Omron CX-Programmer project НовыйПроект (CX-Programmer 9.52)

# PLC НовыйПЛК1: CP1L-E EM

## Global symbols (name address type ; comment)
AbsoluteCounterPoisition D30 DINT  ; Абсолютное значение счетчика импульсов энкодера
AnalogSP D101 CHANNEL  ; Задание скорости с платы аналоговых выходов ПЛК
D1000 CHANNEL  ; выбор адреса ПЧ
D1002 CHANNEL  ; Выбор типа ПЧ - МХ2
T0000 BOOL  ; Бит запуска преобразования в аналоговую форму
AutomaticControl W0.09 BOOL  ; Автоматическое управление
CounterMinDistanceBetweenSaws D42 DINT  ; Минимальное расстояние между пилами в импульсах энкодера
DecButton W18.01 BOOL  ; Кнопка декремента на панели
EndOfCycleInAutomatic W0.13 BOOL  ; Конец цикла автоматического режима
ForwardCommand 100.02 BOOL  ; Команда Вперед на ПЧ
IncButton W18.00 BOOL  ; Кнопка инкремента на панели
InverterReady 0.06 BOOL  ; Частотный преобразователь готов (сигнал с ПЧ)
InverterRunning 0.07 BOOL  ; Частотный преобразователь запущен (сигнал с ПЧ)
LeftLimitSwitch 0.08 BOOL  ; Левый концевик
ManualControl W0.04 BOOL  ; Ручное управление
ManualLeft W0.07 BOOL  ; Влево в ручном режиме
ManualRight W0.08 BOOL  ; Вправо в ручном режиме
MinDistanceBetweenSaws D40 DINT  ; Уставка минимального расстояния между пилами (в крайнем положении)
MoveToPosition W0.03 BOOL  ; Переехать в заданное положение
PID_control1 CoordinateConverting
PV_HighspeedCounter D35 DINT  ; Текущее значение высокоскоростного счетчика
PreviousCounterPosition D32 DINT  ; Предыдущая позиция энкодера
PulseTravelDistance W13 UDINT  ; Число импульсов, необходимое для достижения положения
PulseVelocityInManual W10 UDINT  ; Скорость выдачи импульсов в ручном режиме
ResetPositioningInAutomatic W0.12 BOOL  ; Сброс функции позиционирования из автоматического режима
ResetPositioningInManual W0.11 BOOL  ; Сброс функции позиционирования из ручного режима
ReverseCommand 100.03 BOOL  ; Команда Назад на ПЧ
RightLimitSwitch 0.03 BOOL  ; Правый концевик
SawInLimitPosition W0.06 BOOL  ; Пила в конечном положении
SawSetPosition D11 INT  ; Заданное положение пилы (мм)
SawTravelDirection W0.10 BOOL  ; Направление движения пилы
StartLeftButton W0.00 BOOL  ; $?St$Bk?_#[3] / Кнопка "Пуск влево"$?St$Bk?_#[3]
StartRightButton W0.01 BOOL  ; $?St$Bk?_#[4] / Кнопка "Пуск вправо"$?St$Bk?_#[4]
StopButton W0.02 BOOL  ; $?St$Bk?_#[5] / Кнопка "Стоп"$?St$Bk?_#[5]
SystemReady W0.05 BOOL  ; Система в норме
ПЧ INV002_Refresh_X31_

## Program НоваяЗадача1 (cyclic task 0)
Local symbols
SawTravelDirection1 W0.15 BOOL
UPRmax D200 DINT  ; ограничение управления
Пуск 110.00 BOOL
Реверс 110.01 BOOL

### Section hmi

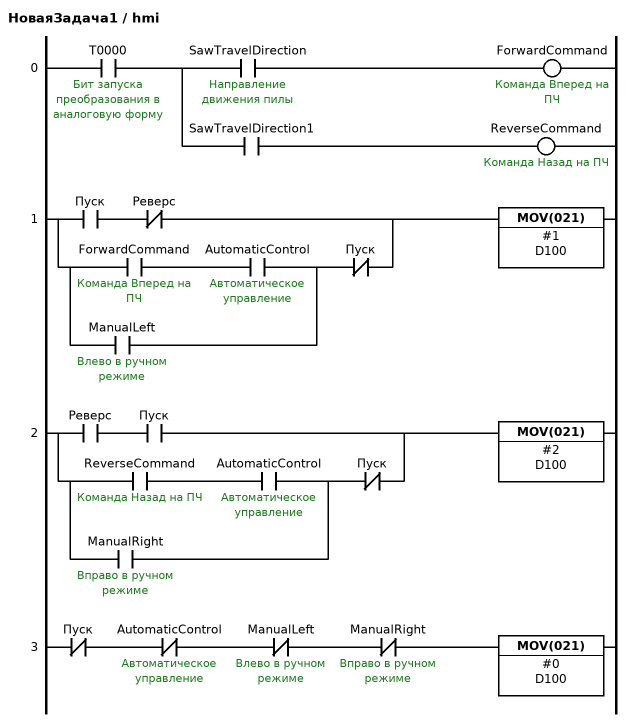
; rung 0
LD T0000  ; Бит запуска преобразования в аналоговую форму
OUT TR0
AND SawTravelDirection  ; Направление движения пилы
OUT ForwardCommand  ; Команда Вперед на ПЧ
LD TR0
AND SawTravelDirection1
OUT ReverseCommand  ; Команда Назад на ПЧ
; rung 1
LD Пуск
ANDNOT Реверс
LD ForwardCommand  ; Команда Вперед на ПЧ
AND AutomaticControl  ; Автоматическое управление
OR ManualLeft  ; Влево в ручном режиме
ANDNOT Пуск
ORLD
MOV(021) #1 D100
; rung 2
LD Реверс
AND Пуск
LD ReverseCommand  ; Команда Назад на ПЧ
AND AutomaticControl  ; Автоматическое управление
OR ManualRight  ; Вправо в ручном режиме
ANDNOT Пуск
ORLD
MOV(021) #2 D100
; rung 3
LDNOT Пуск
ANDNOT AutomaticControl  ; Автоматическое управление
ANDNOT ManualLeft  ; Влево в ручном режиме
ANDNOT ManualRight  ; Вправо в ручном режиме
MOV(021) #0 D100

### Section ModBus

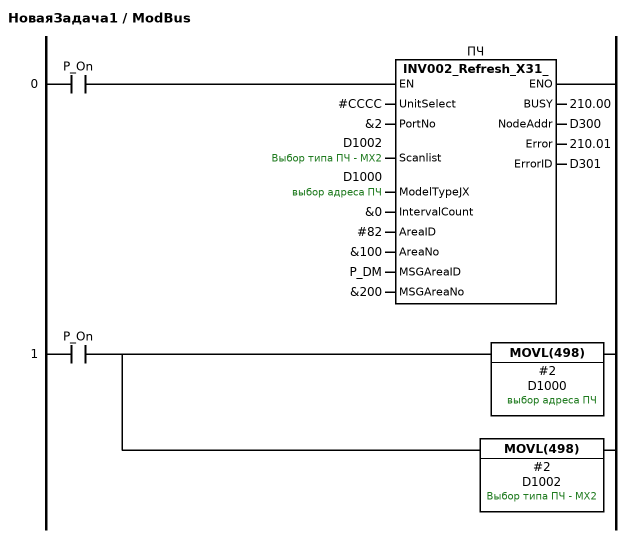
; rung 0
LD P_On
CALL ПЧ : INV002_Refresh_X31_ (UnitSelect := #CCCC, PortNo := &2, Scanlist := D1002, ModelTypeJX := D1000, IntervalCount := &0, AreaID := #82, AreaNo := &100, MSGAreaID := P_DM, MSGAreaNo := &200, BUSY => 210.00, NodeAddr => D300, Error => 210.01, ErrorID => D301)  ; Выбор типа ПЧ - МХ2, выбор адреса ПЧ
; rung 1
LD P_On
MOVL(498) #2 D1000  ; выбор адреса ПЧ
MOVL(498) #2 D1002  ; Выбор типа ПЧ - МХ2

### Section Initialization

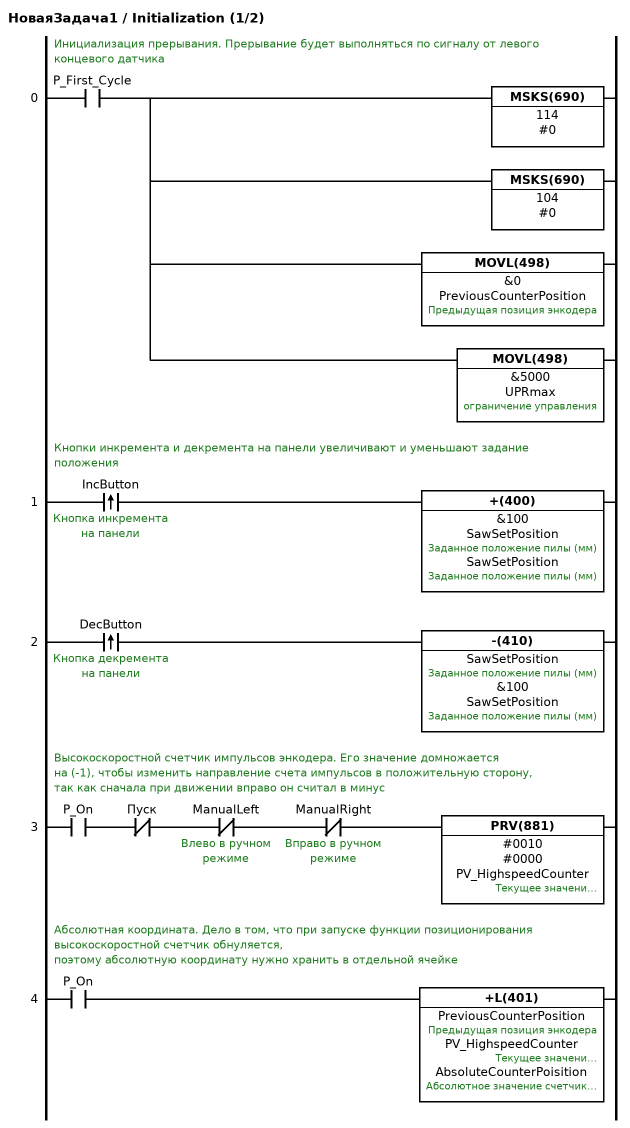
; rung 0: Инициализация прерывания. Прерывание будет выполняться по сигналу от левого концевого датчика
LD P_First_Cycle
MSKS(690) 114 #0
MSKS(690) 104 #0
MOVL(498) &0 PreviousCounterPosition  ; Предыдущая позиция энкодера
MOVL(498) &5000 UPRmax  ; ограничение управления
; rung 1: Кнопки инкремента и декремента на панели увеличивают и уменьшают задание положения
@LD IncButton  ; Кнопка инкремента на панели
+(400) &100 SawSetPosition SawSetPosition  ; Заданное положение пилы (мм)
; rung 2
@LD DecButton  ; Кнопка декремента на панели
-(410) SawSetPosition &100 SawSetPosition  ; Заданное положение пилы (мм)
; rung 3: Высокоскоростной счетчик импульсов энкодера. Его значение домножается / на (-1), чтобы изменить направление счета импульсов в положительную сторону, / так как сначала при движении вправо он считал в минус
LD P_On
ANDNOT Пуск
ANDNOT ManualLeft  ; Влево в ручном режиме
ANDNOT ManualRight  ; Вправо в ручном режиме
PRV(881) #0010 #0000 PV_HighspeedCounter  ; Текущее значение высокоскоростного счетчика
; rung 4: Абсолютная координата. Дело в том, что при запуске функции позиционирования высокоскоростной счетчик обнуляется, / поэтому абсолютную координату нужно хранить в отдельной ячейке
LD P_On
+L(401) PreviousCounterPosition PV_HighspeedCounter AbsoluteCounterPoisition  ; Предыдущая позиция энкодера, Текущее значение высокоскоростного счетчика, Абсолютное значение счетчика импульсов энкодера

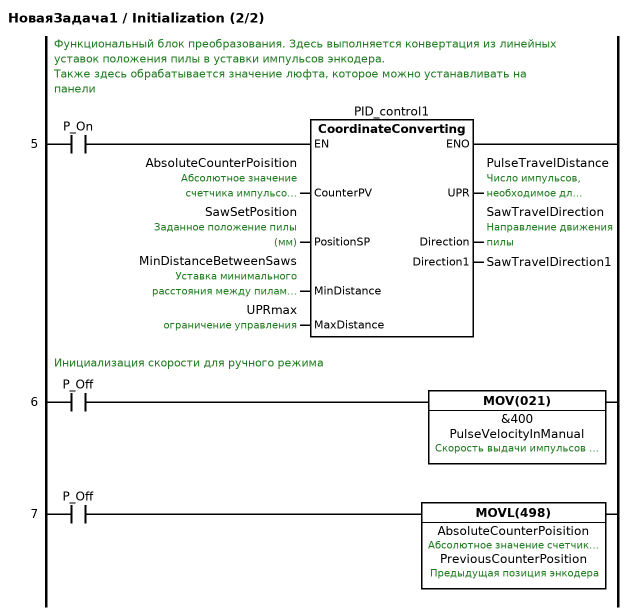
; rung 5: Функциональный блок преобразования. Здесь выполняется конвертация из линейных уставок положения пилы в уставки импульсов энкодера. / Также здесь обрабатывается значение люфта, которое можно устанавливать на панели
LD P_On
CALL PID_control1 : CoordinateConverting (CounterPV := AbsoluteCounterPoisition, PositionSP := SawSetPosition, MinDistance := MinDistanceBetweenSaws, MaxDistance := UPRmax, UPR => PulseTravelDistance, Direction => SawTravelDirection, Direction1 => SawTravelDirection1)  ; Абсолютное значение счетчика импульсов энкодера, Заданное положение пилы (мм), Уставка минимального расстояния между пилами (в крайнем положении), ограничение управления, Число импульсов, необходимое для достижения положения, Направление движения пилы
; rung 6: Инициализация скорости для ручного режима
LD P_Off
MOV(021) &400 PulseVelocityInManual  ; Скорость выдачи импульсов в ручном режиме
; rung 7
LD P_Off
MOVL(498) AbsoluteCounterPoisition PreviousCounterPosition  ; Абсолютное значение счетчика импульсов энкодера, Предыдущая позиция энкодера

### Section Status

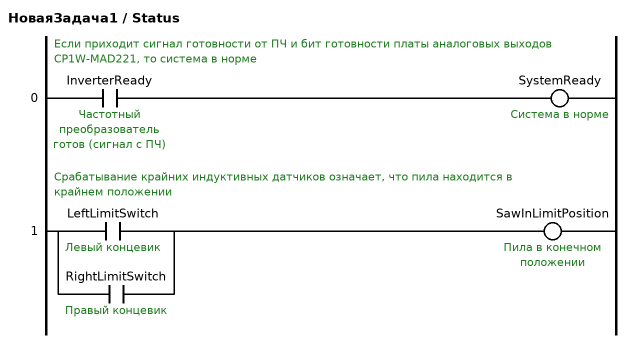
; rung 0: Если приходит сигнал готовности от ПЧ и бит готовности платы аналоговых выходов CP1W-MAD221, то система в норме
LD InverterReady  ; Частотный преобразователь готов (сигнал с ПЧ)
OUT SystemReady  ; Система в норме
; rung 1: Срабатывание крайних индуктивных датчиков означает, что пила находится в крайнем положении
LD LeftLimitSwitch  ; Левый концевик
OR RightLimitSwitch  ; Правый концевик
OUT SawInLimitPosition  ; Пила в конечном положении

### Section ManualControl

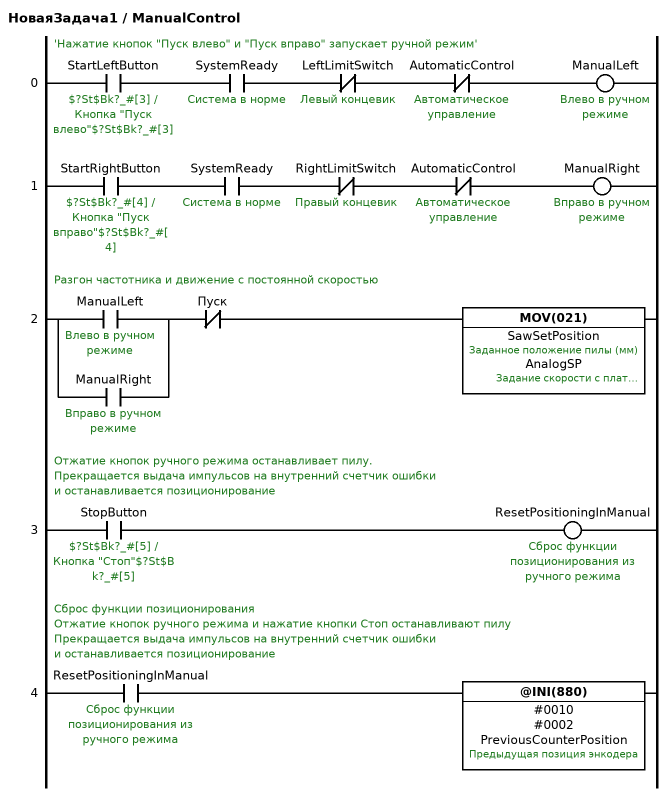
; rung 0: 'Нажатие кнопок "Пуск влево" и "Пуск вправо" запускает ручной режим'
LD StartLeftButton  ; $?St$Bk?_#[3] / Кнопка "Пуск влево"$?St$Bk?_#[3]
AND SystemReady  ; Система в норме
ANDNOT LeftLimitSwitch  ; Левый концевик
ANDNOT AutomaticControl  ; Автоматическое управление
OUT ManualLeft  ; Влево в ручном режиме
; rung 1
LD StartRightButton  ; $?St$Bk?_#[4] / Кнопка "Пуск вправо"$?St$Bk?_#[4]
AND SystemReady  ; Система в норме
ANDNOT RightLimitSwitch  ; Правый концевик
ANDNOT AutomaticControl  ; Автоматическое управление
OUT ManualRight  ; Вправо в ручном режиме
; rung 2: Разгон частотника и движение с постоянной скоростью
LD ManualLeft  ; Влево в ручном режиме
OR ManualRight  ; Вправо в ручном режиме
ANDNOT Пуск
MOV(021) SawSetPosition AnalogSP  ; Заданное положение пилы (мм), Задание скорости с платы аналоговых выходов ПЛК
; rung 3: Отжатие кнопок ручного режима останавливает пилу. / Прекращается выдача импульсов на внутренний счетчик ошибки / и останавливается позиционирование
LD StopButton  ; $?St$Bk?_#[5] / Кнопка "Стоп"$?St$Bk?_#[5]
OUT ResetPositioningInManual  ; Сброс функции позиционирования из ручного режима
; rung 4: Сброс функции позиционирования / Отжатие кнопок ручного режима и нажатие кнопки Стоп останавливают пилу / Прекращается выдача импульсов на внутренний счетчик ошибки / и останавливается позиционирование
LD ResetPositioningInManual  ; Сброс функции позиционирования из ручного режима
@INI(880) #0010 #0002 PreviousCounterPosition  ; Предыдущая позиция энкодера

### Section AutomaticControl

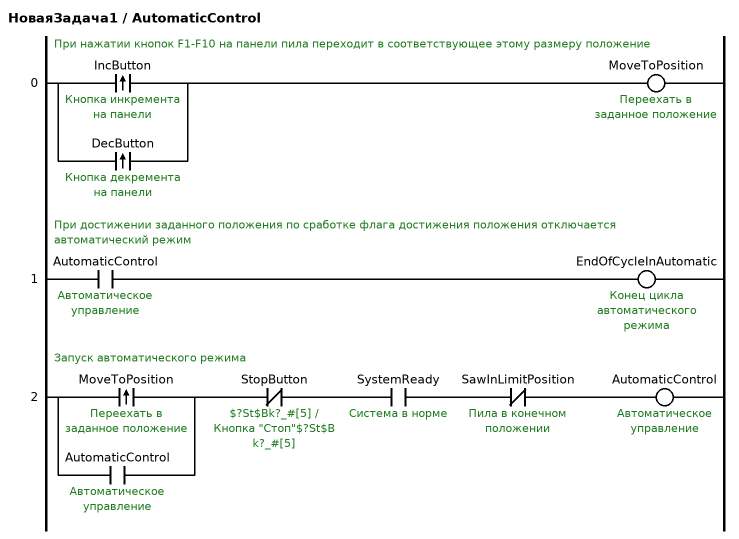
; rung 0: При нажатии кнопок F1-F10 на панели пила переходит в соответствующее этому размеру положение
@LD IncButton  ; Кнопка инкремента на панели
@OR DecButton  ; Кнопка декремента на панели
OUT MoveToPosition  ; Переехать в заданное положение
; rung 1: При достижении заданного положения по сработке флага достижения положения отключается автоматический режим
LD AutomaticControl  ; Автоматическое управление
OUT EndOfCycleInAutomatic  ; Конец цикла автоматического режима
; rung 2: Запуск автоматического режима
@LD MoveToPosition  ; Переехать в заданное положение
OR AutomaticControl  ; Автоматическое управление
ANDNOT StopButton  ; $?St$Bk?_#[5] / Кнопка "Стоп"$?St$Bk?_#[5]
AND SystemReady  ; Система в норме
ANDNOT SawInLimitPosition  ; Пила в конечном положении
OUT AutomaticControl  ; Автоматическое управление

### Section Inverter

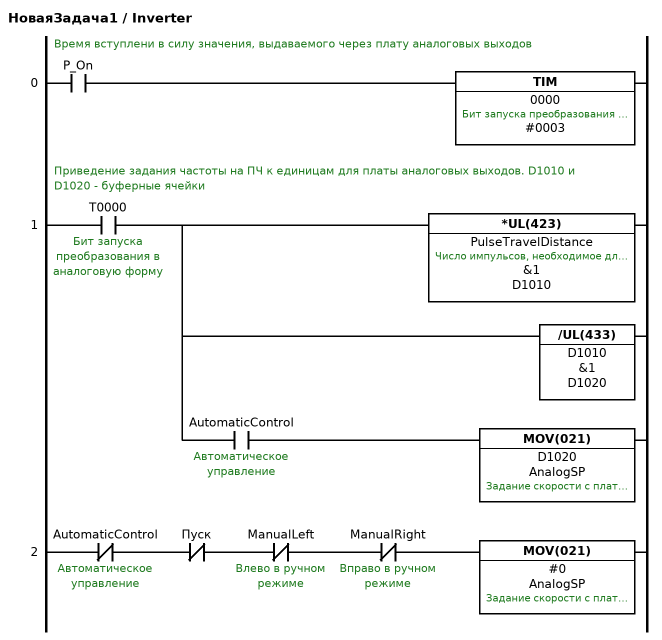
; rung 0: Время вступлени в силу значения, выдаваемого через плату аналоговых выходов
LD P_On
TIM 0000 #0003  ; Бит запуска преобразования в аналоговую форму
; rung 1: Приведение задания частоты на ПЧ к единицам для платы аналоговых выходов. D1010 и D1020 - буферные ячейки
LD T0000  ; Бит запуска преобразования в аналоговую форму
*UL(423) PulseTravelDistance &1 D1010  ; Число импульсов, необходимое для достижения положения
/UL(433) D1010 &1 D1020
AND AutomaticControl  ; Автоматическое управление
MOV(021) D1020 AnalogSP  ; Задание скорости с платы аналоговых выходов ПЛК
; rung 2
LDNOT AutomaticControl  ; Автоматическое управление
ANDNOT Пуск
ANDNOT ManualLeft  ; Влево в ручном режиме
ANDNOT ManualRight  ; Вправо в ручном режиме
MOV(021) #0 AnalogSP  ; Задание скорости с платы аналоговых выходов ПЛК

### Section END
; rung 0
END(001)

## Program LimitSwitch (interrupt task 144)

### Section CounterResetting

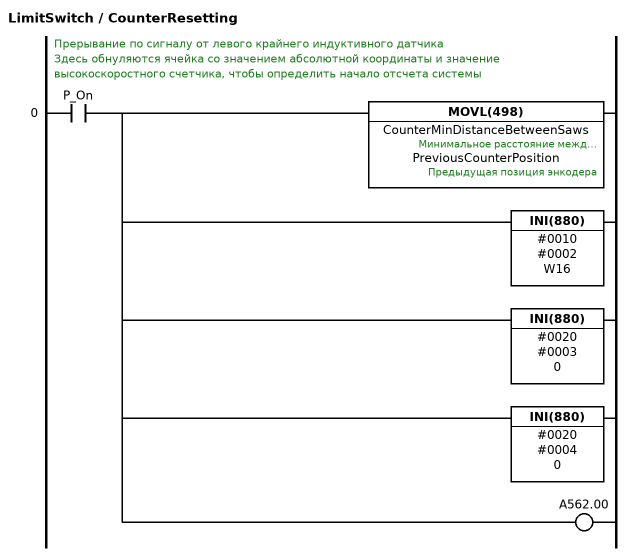
; rung 0: Прерывание по сигналу от левого крайнего индуктивного датчика / Здесь обнуляются ячейка со значением абсолютной координаты и значение / высокоскоростного счетчика, чтобы определить начало отсчета системы
LD P_On
MOVL(498) CounterMinDistanceBetweenSaws PreviousCounterPosition  ; Минимальное расстояние между пилами в импульсах энкодера, Предыдущая позиция энкодера
INI(880) #0010 #0002 W16
INI(880) #0020 #0003 0
INI(880) #0020 #0004 0
OUT A562.00

### Section END
; rung 0
END(001)

## Function block CoordinateConverting
VAR_INPUT
  CounterPV : DINT;
  PositionSP : INT;
  MinDistance : DINT := 10;
  MaxDistance : DINT := 5000;
END_VAR
VAR_OUTPUT
  UPR : DINT;
  CounterSP : DINT;
  Direction : BOOL;
  TravelDistance : DINT;
  Direction1 : BOOL;
END_VAR
VAR
  TravelDistance0 : DINT;
  Ki : DINT := 20;
END_VAR
CounterSP := INT_TO_DINT(PositionSP);
TravelDistance :=(CounterSP - CounterPV);                               (*ошибка позиции*)
UPR := TravelDistance+Ki* (TravelDistance- TravelDistance0);  (*приращение управления*)
IF ((UPR) < 0)
	THEN 
	 Direction := TRUE; Direction1:=FALSE;
	 ELSE Direction := FALSE; Direction1:=TRUE;
	END_IF;
IF (ABS(CounterSP -CounterPV) >ABS(MinDistance))           (*зона нечуствительности*)
	THEN UPR :=(ABS(UPR));
ELSE UPR := 0; Direction := FALSE;Direction1 := FALSE;
END_IF; 
IF (ABS(UPR) >ABS(MaxDistance))
	THEN UPR :=(ABS(MaxDistance));
ELSE UPR :=ABS(UPR);
END_IF; 
TravelDistance0 := TravelDistance;

## Function block INV002_Refresh_X31_
; <Status Refresh>Refreshes inverter status.
VAR_INPUT
  UnitSelect : INT;  (* Specify the connetcted Unit SCB=#BBBB_SCU=&0to&15 *)
  PortNo : INT := 1;  (* Serial port No. &0to&2 *)
  Scanlist : DWORD;  (* Scanlist *)
  ModelTypeJX : DWORD;  (* JX/MX or MX2/RX Classification for older Inverter types also this Bit has to be set, like scanlist *)
  IntervalCount : UINT;  (* Interval *)
  AreaID : WORD;  (* Using Area Classification *)
  AreaNo : INT;  (* Using Area Number *)
  MSGAreaID : WORD;  (* Message Area Classification *)
  MSGAreaNo : INT;  (* Message Area Number *)
END_VAR
VAR_OUTPUT
  BUSY : BOOL;  (* Processing Flag 0:Transferring Complete 1:Transferring *)
  NodeAddr : INT;  (* Executing Axis Number *)
  Error : BOOL;  (* Error *)
  ErrorID : WORD;  (* Error Code *)
END_VAR
VAR
  WAIT : BOOL;  (* First Cycle Wait Bit *)
  UnitSelect_Tmp : INT;  (* SCB/Select SCU Bit storage(internal variables) *)
  Type_W AT W0 : WORD;  (* Address type WR start address *)
  Type_Io AT 0 : WORD;  (* Address type IO start address *)
  Type_H AT H0 : WORD;  (* Address type HR start address *)
  Type_D AT D0 : WORD;  (* Address type DM start address *)
  Tmp_IR : ARRAY[0..3] OF DINT;  (* Temporary IR for internal variables *)
  Tmp_Data : ARRAY[0..30] OF WORD;  (* For internal Calculation *)
  Time_Value : UINT;  (* Interval Check Time Present Value *)
  Status_Inv_No : INT;  (* Status Command Slave Number *)
  Status_Commmnd_INT : BOOL;  (* Status Interrupt Flag *)
  Status_Commmnd_Enable : BOOL;  (* Enable Execution Status Command *)
  Status_2Cp : WORD;  (* second word of coils beginning with coil 1F to 2E *)
  Status_2C : WORD;  (* Register 2C Response Data *)
  Set_IR AT 0 : WORD;  (* Index register temporary setting *)
  Scanlist_Tmp : DWORD;  (* Scanlist storage *)
  SaveIR : ARRAY[0..3] OF DINT;  (* IR0toIR3 *)
  SaveDR : WORD;  (* DR0 *)
  Response_NG : BOOL;  (* Response error *)
  Response_Data : ARRAY[0..20] OF WORD;  (* CMND response data *)
  Response_CodeNG : BOOL;  (* Response end code error *)
  PortNo_Tmp : INT;  (* Serial port No. storage(internal variables) *)
  Phase : WORD;  (* Process Procedure *)
  P_FreeRunningCounter_10 AT A0 : UINT;  (* 10ms free running incremental counter *)
  P_Error : BOOL;  (* Error Flag *)
  P_EM_MaxNo AT A338 : INT;  (* EM bank size *)
  P_ComPort_WatchResTime AT A581 : INT;  (* FB Communications command response Monitor time *)
  P_ComPort_Retry AT A580 : WORD;  (* FB Communications command retry count *)
  P_ComPort_Finished0_7 AT A214 : WORD;  (* Communications Complete Cycle Bit *)
  P_ComPort_AutoAlloc_Available AT A202.15 : BOOL;  (* Auto allocation avarable bit *)
  P_ComPort_AllocatedNumber AT A218 : INT;  (* Network port No. *)
  Ok_WR : BOOL;  (* Selected WR area range OK *)
  Ok_IO : BOOL;  (* Selected CIO area range OK *)
  Ok_HR : BOOL;  (* Selected HR area range OK *)
  Ok_EM : BOOL;  (* Selected EM area range OK *)
  Ok_DM : BOOL;  (* Selected DM area range OK *)
  Ok_Bit : BOOL;  (* Range Check OK Bit *)
  Offset : DINT;  (* For Address Culcurate *)
  No : INT;  (* MatrixNo *)
  NG_Bit : BOOL;  (* Range Check NG Bit *)
  MSGAreaNo_Tmp : INT;  (* Message Area Number storage(internal variables) *)
  MSGAreaID_Tmp : WORD;  (* Message Area Classification storage(internal variables) *)
  ModelTypeMV_Tmp : DWORD;  (* MV/RVClassification storage(internal variables) *)
  Message_Command_Done : BOOL;  (* Exist Message Command Flag *)
  Last_Area_Status : ARRAY[0..61] OF WORD;  (* The Last Time IOM Status Condition *)
  Inv_Use_Count : INT;  (* Amount of Use Inverter Number *)
  Inv_Status_Count : INT;  (* Inverter Status Command Execution Number *)
  Inv_NodeArea : ARRAY[0..31] OF WORD;  (* Applicable Axis Inverter Model and Number Store Area *)
  INV_Error : BOOL;  (* Inverter Error *)
  Inv_Command_Change_Position : INT;  (* Inverter Write Command Changing Position *)
  IntervalCount_Tmp : UINT;  (* Interval storage(internal variables) *)
  IntervalCount_Compare : INT;  (* IntervalCompare Value *)
  Interval_TimeUp : BOOL;  (* Interval Time Up *)
  Interval_Start : BOOL;  (* Interval Count Start *)
  FreeRunningCounter_Tmp : UINT;  (* 10ms free running incremental counter record *)
  Error_Skip : BOOL;  (* Fatal Error Skip Flag *)
  EM_NoCheck : INT;  (* EM bank size check area *)
  Directive_Data : ARRAY[0..1] OF WORD;  (* Command data *)
  Data_Change : BOOL;  (* Detect input data change *)
  Control_Data : ARRAY[0..5] OF WORD;  (* CMND control data *)
  Command_Fin : BOOL;  (* CMND Transferring End *)
  Command_Data_Change2 : BOOL;
  Command_Data_Change : BOOL;  (* Write Command Data Changing *)
  Command_Data : ARRAY[0..21] OF WORD;  (* CMND command data *)
  Command_CheckNo : INT;  (* Write Command Check Complete Number *)
  CMNDPort : INT;  (* Port Number 1(Automatic Setting) *)
  BUSY_Run : BOOL;  (* Internal Processing Flag *)
  AreaNo_Tmp : INT;  (* Using Area Number storage(internal variables) *)
  AreaID_Tmp : WORD;  (* Using Area Classification storage(internal variables) *)
  AddressOk_Bit : BOOL;  (* Addrss Range Check OK Bit *)
  maxindex : UINT;  (* maximum possible inverters *)
  index : UINT;  (* index in the for next loop *)
  controlw : WORD;  (* controlword *)
  index2 : UINT;
  index3 : UINT;
  index4 : INT;  (* = index + 16 *)
  index5 : INT;  (* = index + 16 *)
  index6 : INT;  (* index3 +32 *)
  index7 : INT;
  Inv_Type_RX : BOOL;
END_VAR

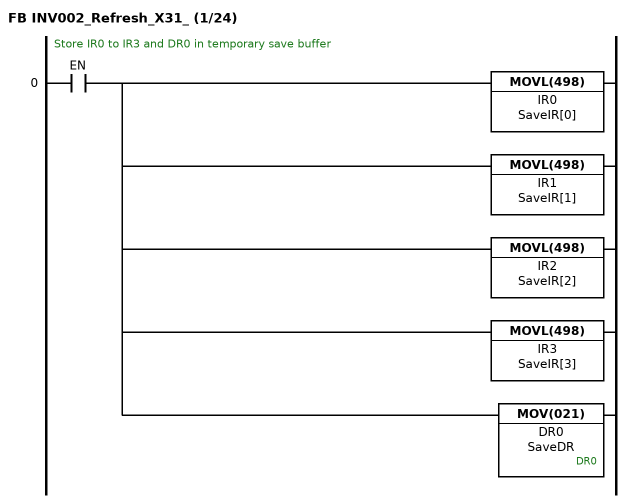
; rung 0: Store IR0 to IR3 and DR0 in temporary save buffer
LD EN
MOVL(498) IR0 SaveIR[0]
MOVL(498) IR1 SaveIR[1]
MOVL(498) IR2 SaveIR[2]
MOVL(498) IR3 SaveIR[3]
MOV(021) DR0 SaveDR  ; DR0

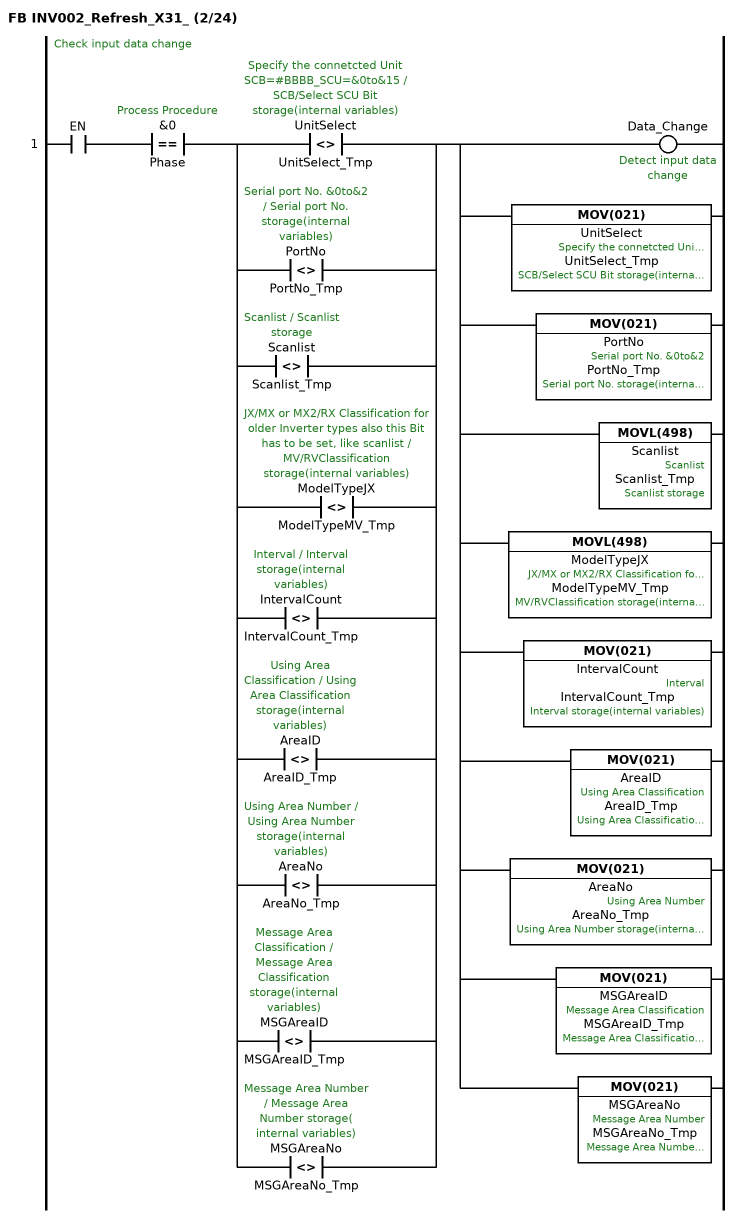
; rung 1: Check input data change
LD EN
AND=(300) &0 Phase  ; Process Procedure
LD<>(305) UnitSelect UnitSelect_Tmp  ; Specify the connetcted Unit SCB=#BBBB_SCU=&0to&15, SCB/Select SCU Bit storage(internal variables)
OR<>(305) PortNo PortNo_Tmp  ; Serial port No. &0to&2, Serial port No. storage(internal variables)
OR<>L(306) Scanlist Scanlist_Tmp  ; Scanlist, Scanlist storage
OR<>L(306) ModelTypeJX ModelTypeMV_Tmp  ; JX/MX or MX2/RX Classification for older Inverter types also this Bit has to be set, like scanlist, MV/RVClassification storage(internal variables)
OR<>(305) IntervalCount IntervalCount_Tmp  ; Interval, Interval storage(internal variables)
OR<>(305) AreaID AreaID_Tmp  ; Using Area Classification, Using Area Classification storage(internal variables)
OR<>(305) AreaNo AreaNo_Tmp  ; Using Area Number, Using Area Number storage(internal variables)
OR<>(305) MSGAreaID MSGAreaID_Tmp  ; Message Area Classification, Message Area Classification storage(internal variables)
OR<>(305) MSGAreaNo MSGAreaNo_Tmp  ; Message Area Number, Message Area Number storage(internal variables)
ANDLD
OUT Data_Change  ; Detect input data change
MOV(021) UnitSelect UnitSelect_Tmp  ; Specify the connetcted Unit SCB=#BBBB_SCU=&0to&15, SCB/Select SCU Bit storage(internal variables)
MOV(021) PortNo PortNo_Tmp  ; Serial port No. &0to&2, Serial port No. storage(internal variables)
MOVL(498) Scanlist Scanlist_Tmp  ; Scanlist, Scanlist storage
MOVL(498) ModelTypeJX ModelTypeMV_Tmp  ; JX/MX or MX2/RX Classification for older Inverter types also this Bit has to be set, like scanlist, MV/RVClassification storage(internal variables)
MOV(021) IntervalCount IntervalCount_Tmp  ; Interval, Interval storage(internal variables)
MOV(021) AreaID AreaID_Tmp  ; Using Area Classification, Using Area Classification storage(internal variables)
MOV(021) AreaNo AreaNo_Tmp  ; Using Area Number, Using Area Number storage(internal variables)
MOV(021) MSGAreaID MSGAreaID_Tmp  ; Message Area Classification, Message Area Classification storage(internal variables)
MOV(021) MSGAreaNo MSGAreaNo_Tmp  ; Message Area Number, Message Area Number storage(internal variables)

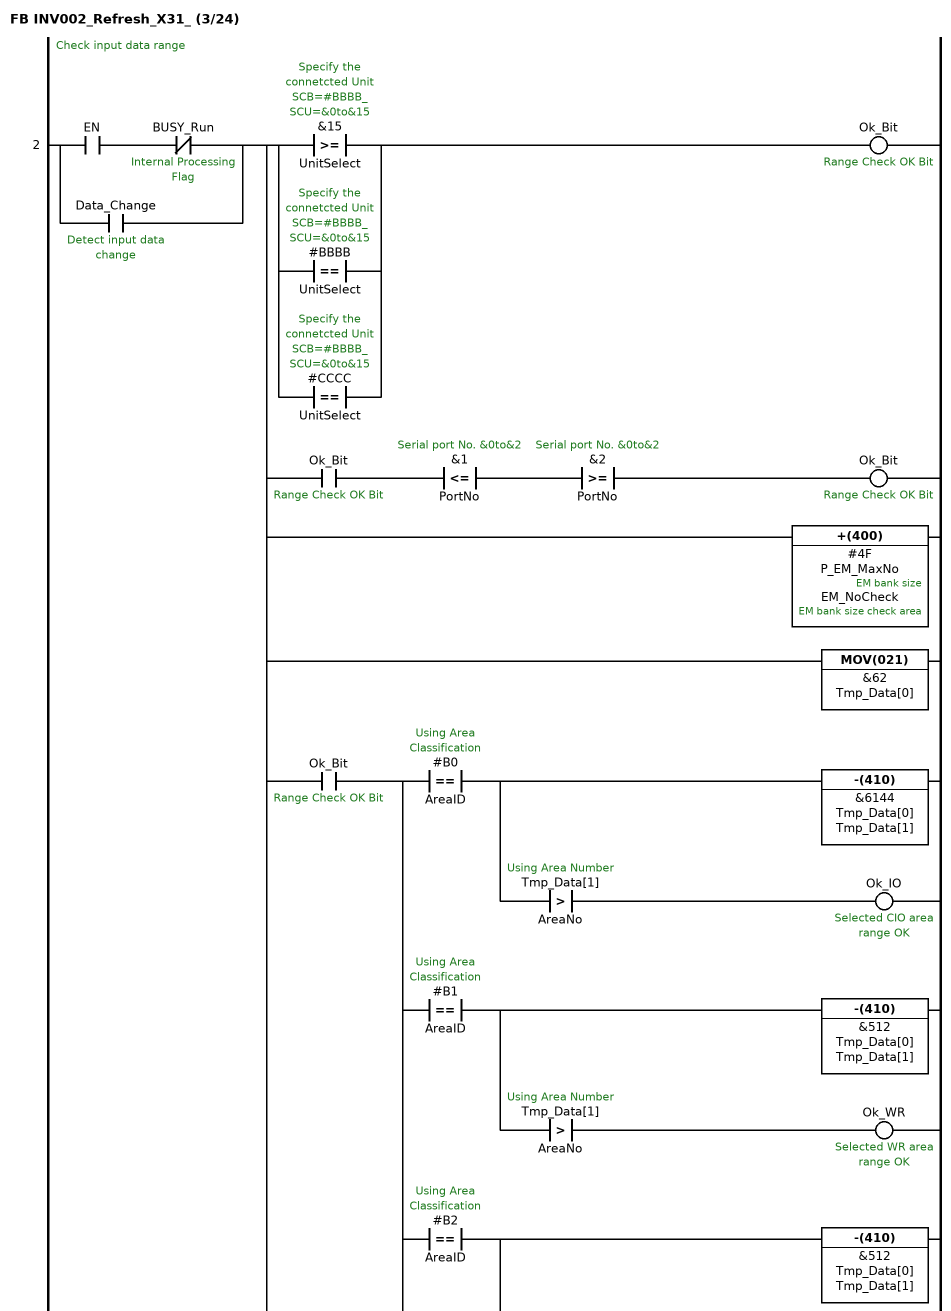

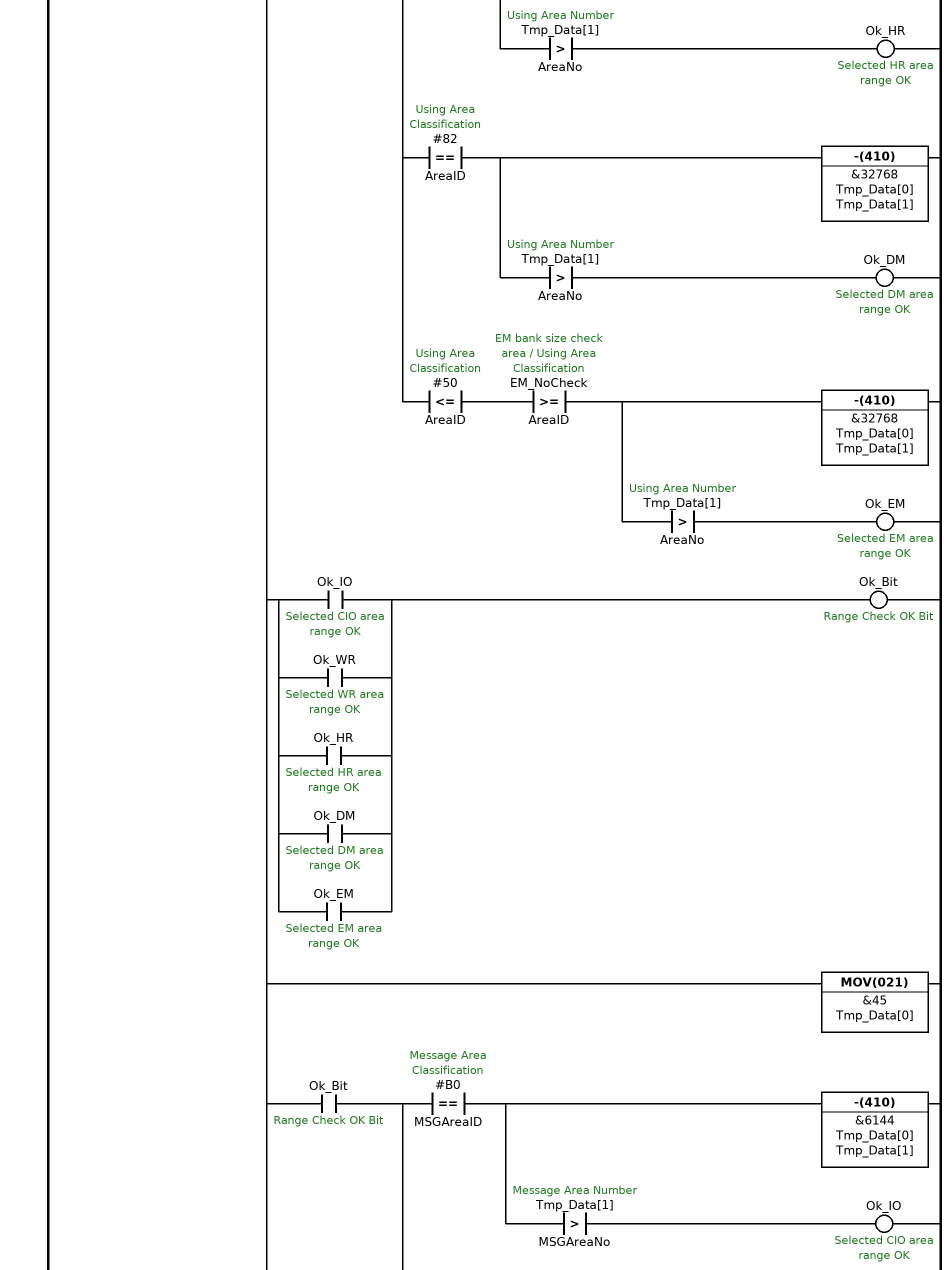

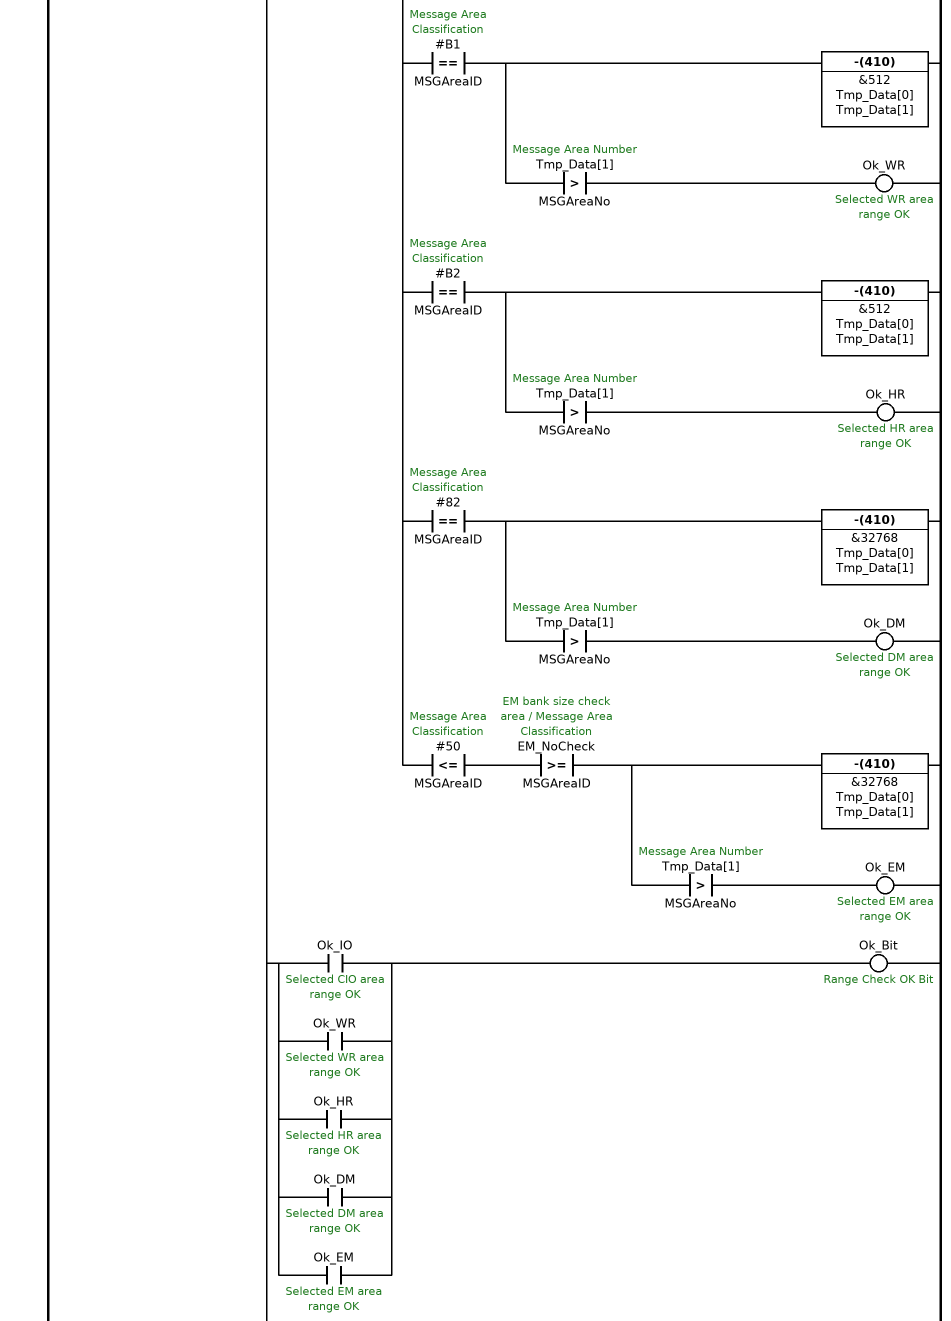

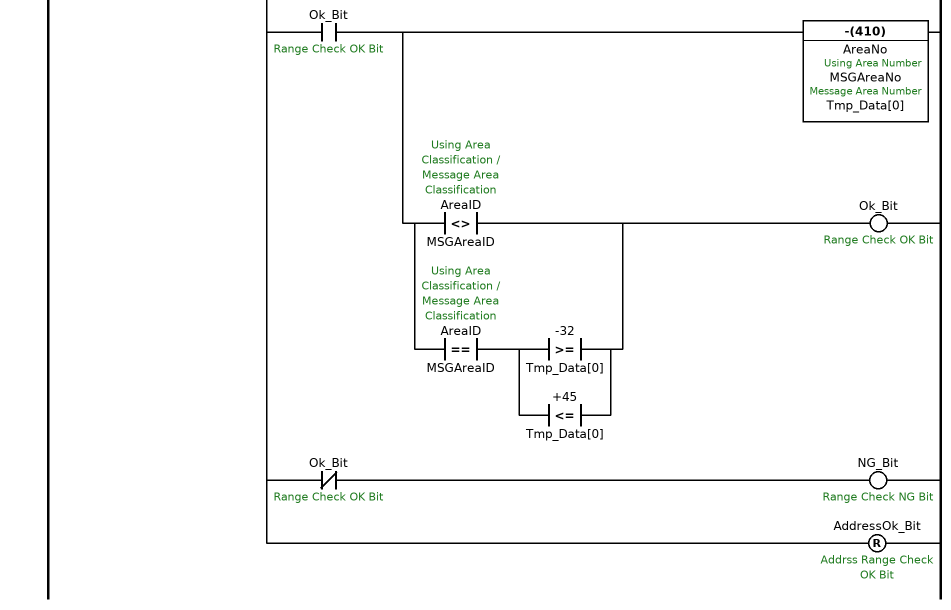
; rung 2: Check input data range
LD EN
ANDNOT BUSY_Run  ; Internal Processing Flag
OR Data_Change  ; Detect input data change
OUT TR0
LD>=(325) &15 UnitSelect  ; Specify the connetcted Unit SCB=#BBBB_SCU=&0to&15
OR=(300) #BBBB UnitSelect  ; Specify the connetcted Unit SCB=#BBBB_SCU=&0to&15
OR=(300) #CCCC UnitSelect  ; Specify the connetcted Unit SCB=#BBBB_SCU=&0to&15
ANDLD
OUT Ok_Bit  ; Range Check OK Bit
LD TR0
AND Ok_Bit  ; Range Check OK Bit
AND<=(315) &1 PortNo  ; Serial port No. &0to&2
AND>=(325) &2 PortNo  ; Serial port No. &0to&2
OUT Ok_Bit  ; Range Check OK Bit
LD TR0
+(400) #4F P_EM_MaxNo EM_NoCheck  ; EM bank size, EM bank size check area
MOV(021) &62 Tmp_Data[0]
AND Ok_Bit  ; Range Check OK Bit
OUT TR1
AND=(300) #B0 AreaID  ; Using Area Classification
-(410) &6144 Tmp_Data[0] Tmp_Data[1]
AND>(320) Tmp_Data[1] AreaNo  ; Using Area Number
OUT Ok_IO  ; Selected CIO area range OK
LD TR1
AND=(300) #B1 AreaID  ; Using Area Classification
-(410) &512 Tmp_Data[0] Tmp_Data[1]
AND>(320) Tmp_Data[1] AreaNo  ; Using Area Number
OUT Ok_WR  ; Selected WR area range OK
LD TR1
AND=(300) #B2 AreaID  ; Using Area Classification
-(410) &512 Tmp_Data[0] Tmp_Data[1]
AND>(320) Tmp_Data[1] AreaNo  ; Using Area Number
OUT Ok_HR  ; Selected HR area range OK
LD TR1
AND=(300) #82 AreaID  ; Using Area Classification
-(410) &32768 Tmp_Data[0] Tmp_Data[1]
AND>(320) Tmp_Data[1] AreaNo  ; Using Area Number
OUT Ok_DM  ; Selected DM area range OK
LD TR1
AND<=(315) #50 AreaID  ; Using Area Classification
AND>=(325) EM_NoCheck AreaID  ; EM bank size check area, Using Area Classification
-(410) &32768 Tmp_Data[0] Tmp_Data[1]
AND>(320) Tmp_Data[1] AreaNo  ; Using Area Number
OUT Ok_EM  ; Selected EM area range OK
LD TR0
LD Ok_IO  ; Selected CIO area range OK
OR Ok_WR  ; Selected WR area range OK
OR Ok_HR  ; Selected HR area range OK
OR Ok_DM  ; Selected DM area range OK
OR Ok_EM  ; Selected EM area range OK
ANDLD
OUT Ok_Bit  ; Range Check OK Bit
LD TR0
MOV(021) &45 Tmp_Data[0]
AND Ok_Bit  ; Range Check OK Bit
OUT TR2
AND=(300) #B0 MSGAreaID  ; Message Area Classification
-(410) &6144 Tmp_Data[0] Tmp_Data[1]
AND>(320) Tmp_Data[1] MSGAreaNo  ; Message Area Number
OUT Ok_IO  ; Selected CIO area range OK
LD TR2
AND=(300) #B1 MSGAreaID  ; Message Area Classification
-(410) &512 Tmp_Data[0] Tmp_Data[1]
AND>(320) Tmp_Data[1] MSGAreaNo  ; Message Area Number
OUT Ok_WR  ; Selected WR area range OK
LD TR2
AND=(300) #B2 MSGAreaID  ; Message Area Classification
-(410) &512 Tmp_Data[0] Tmp_Data[1]
AND>(320) Tmp_Data[1] MSGAreaNo  ; Message Area Number
OUT Ok_HR  ; Selected HR area range OK
LD TR2
AND=(300) #82 MSGAreaID  ; Message Area Classification
-(410) &32768 Tmp_Data[0] Tmp_Data[1]
AND>(320) Tmp_Data[1] MSGAreaNo  ; Message Area Number
OUT Ok_DM  ; Selected DM area range OK
LD TR2
AND<=(315) #50 MSGAreaID  ; Message Area Classification
AND>=(325) EM_NoCheck MSGAreaID  ; EM bank size check area, Message Area Classification
-(410) &32768 Tmp_Data[0] Tmp_Data[1]
AND>(320) Tmp_Data[1] MSGAreaNo  ; Message Area Number
OUT Ok_EM  ; Selected EM area range OK
LD TR0
LD Ok_IO  ; Selected CIO area range OK
OR Ok_WR  ; Selected WR area range OK
OR Ok_HR  ; Selected HR area range OK
OR Ok_DM  ; Selected DM area range OK
OR Ok_EM  ; Selected EM area range OK
ANDLD
OUT Ok_Bit  ; Range Check OK Bit
LD TR0
AND Ok_Bit  ; Range Check OK Bit
-(410) AreaNo MSGAreaNo Tmp_Data[0]  ; Using Area Number, Message Area Number
LD<>(305) AreaID MSGAreaID  ; Using Area Classification, Message Area Classification
LD=(300) AreaID MSGAreaID  ; Using Area Classification, Message Area Classification
LD>=S(327) -32 Tmp_Data[0]
OR<=S(317) +45 Tmp_Data[0]
ANDLD
ORLD
ANDLD
OUT Ok_Bit  ; Range Check OK Bit
LD TR0
ANDNOT Ok_Bit  ; Range Check OK Bit
OUT NG_Bit  ; Range Check NG Bit
LD TR0
RSET AddressOk_Bit  ; Addrss Range Check OK Bit

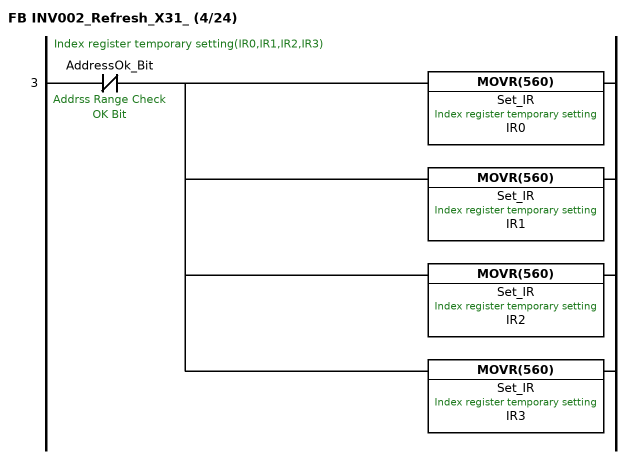
; rung 3: Index register temporary setting(IR0,IR1,IR2,IR3)
LDNOT AddressOk_Bit  ; Addrss Range Check OK Bit
MOVR(560) Set_IR IR0  ; Index register temporary setting
MOVR(560) Set_IR IR1  ; Index register temporary setting
MOVR(560) Set_IR IR2  ; Index register temporary setting
MOVR(560) Set_IR IR3  ; Index register temporary setting

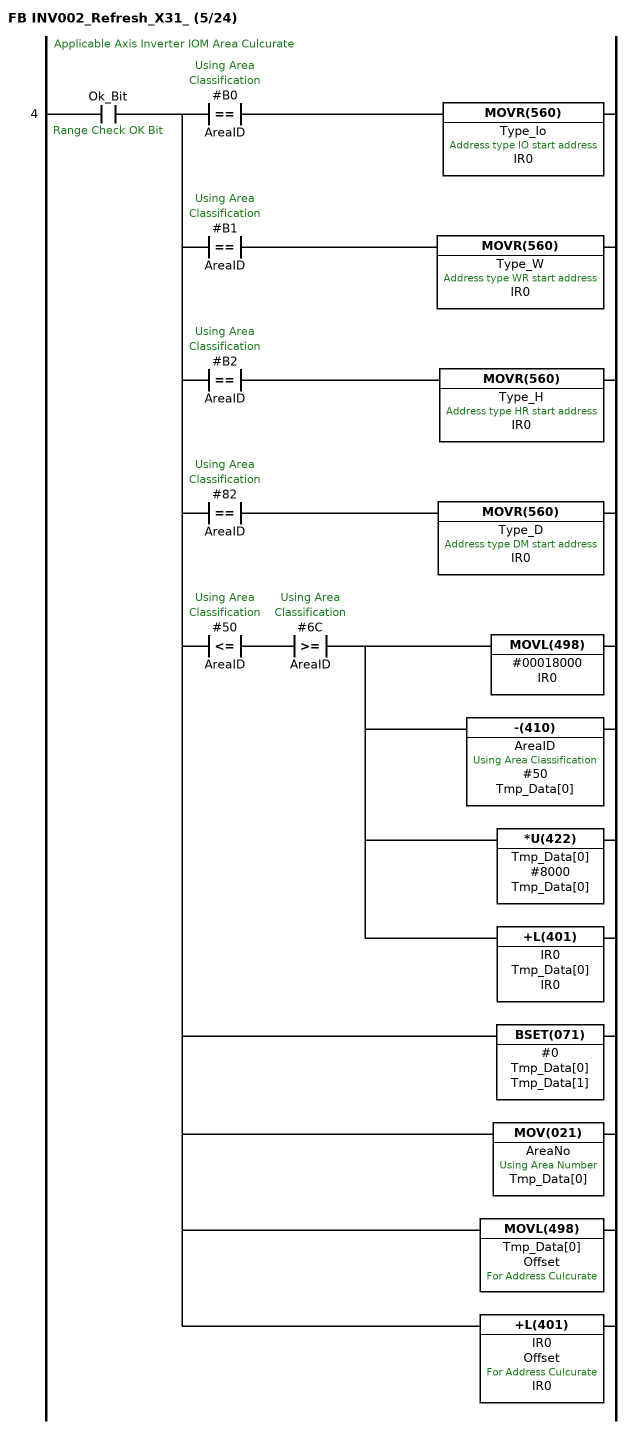
; rung 4: Applicable Axis Inverter IOM Area Culcurate
LD Ok_Bit  ; Range Check OK Bit
OUT TR0
AND=(300) #B0 AreaID  ; Using Area Classification
MOVR(560) Type_Io IR0  ; Address type IO start address
LD TR0
AND=(300) #B1 AreaID  ; Using Area Classification
MOVR(560) Type_W IR0  ; Address type WR start address
LD TR0
AND=(300) #B2 AreaID  ; Using Area Classification
MOVR(560) Type_H IR0  ; Address type HR start address
LD TR0
AND=(300) #82 AreaID  ; Using Area Classification
MOVR(560) Type_D IR0  ; Address type DM start address
LD TR0
AND<=(315) #50 AreaID  ; Using Area Classification
AND>=(325) #6C AreaID  ; Using Area Classification
MOVL(498) #00018000 IR0
-(410) AreaID #50 Tmp_Data[0]  ; Using Area Classification
*U(422) Tmp_Data[0] #8000 Tmp_Data[0]
+L(401) IR0 Tmp_Data[0] IR0
LD TR0
BSET(071) #0 Tmp_Data[0] Tmp_Data[1]
MOV(021) AreaNo Tmp_Data[0]  ; Using Area Number
MOVL(498) Tmp_Data[0] Offset  ; For Address Culcurate
+L(401) IR0 Offset IR0  ; For Address Culcurate

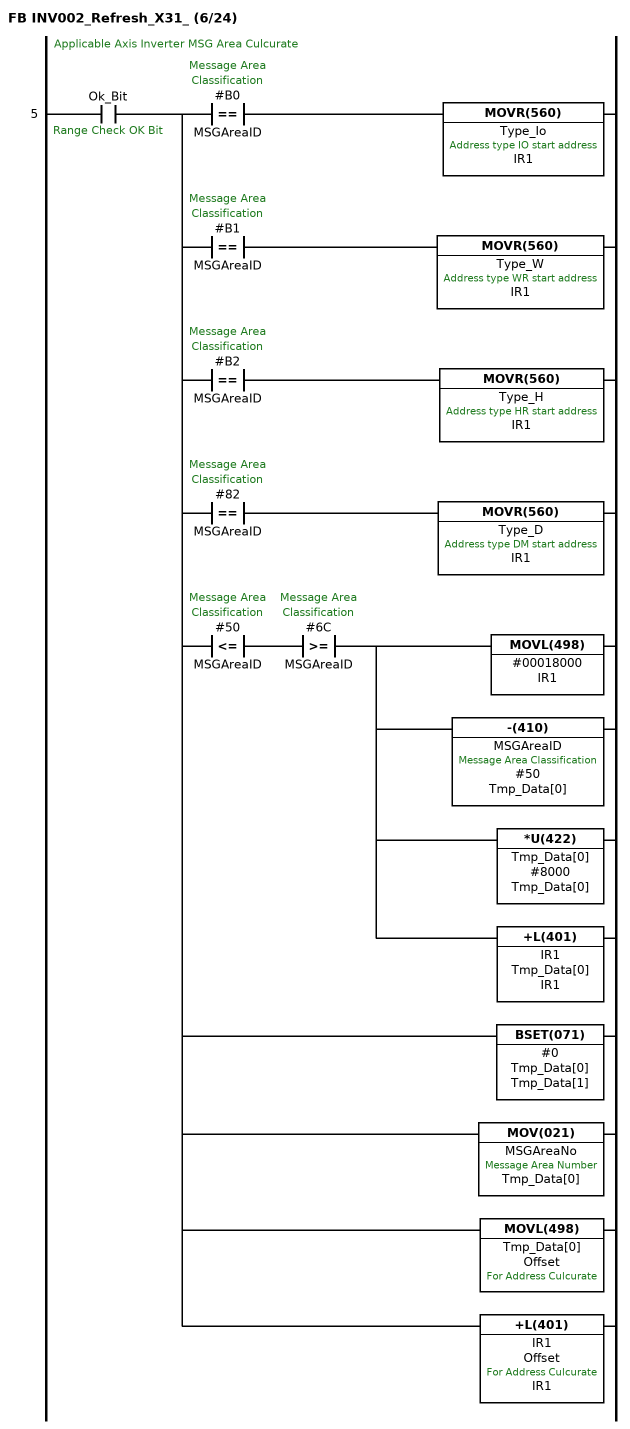
; rung 5: Applicable Axis Inverter MSG Area Culcurate
LD Ok_Bit  ; Range Check OK Bit
OUT TR0
AND=(300) #B0 MSGAreaID  ; Message Area Classification
MOVR(560) Type_Io IR1  ; Address type IO start address
LD TR0
AND=(300) #B1 MSGAreaID  ; Message Area Classification
MOVR(560) Type_W IR1  ; Address type WR start address
LD TR0
AND=(300) #B2 MSGAreaID  ; Message Area Classification
MOVR(560) Type_H IR1  ; Address type HR start address
LD TR0
AND=(300) #82 MSGAreaID  ; Message Area Classification
MOVR(560) Type_D IR1  ; Address type DM start address
LD TR0
AND<=(315) #50 MSGAreaID  ; Message Area Classification
AND>=(325) #6C MSGAreaID  ; Message Area Classification
MOVL(498) #00018000 IR1
-(410) MSGAreaID #50 Tmp_Data[0]  ; Message Area Classification
*U(422) Tmp_Data[0] #8000 Tmp_Data[0]
+L(401) IR1 Tmp_Data[0] IR1
LD TR0
BSET(071) #0 Tmp_Data[0] Tmp_Data[1]
MOV(021) MSGAreaNo Tmp_Data[0]  ; Message Area Number
MOVL(498) Tmp_Data[0] Offset  ; For Address Culcurate
+L(401) IR1 Offset IR1  ; For Address Culcurate

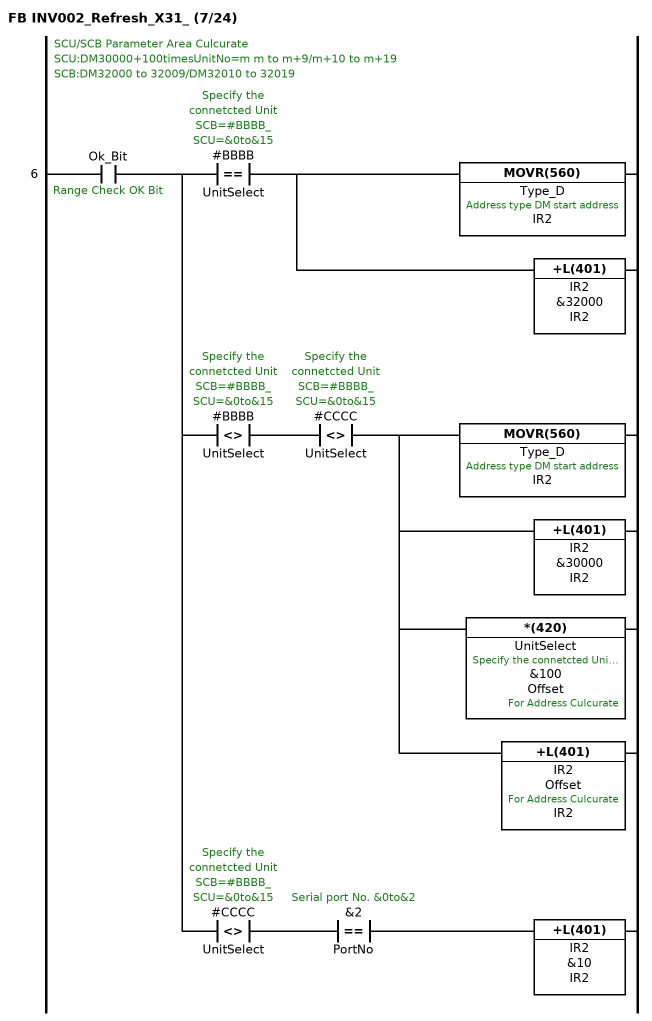
; rung 6: SCU/SCB Parameter Area Culcurate / SCU:DM30000+100timesUnitNo=m m to m+9/m+10 to m+19 / SCB:DM32000 to 32009/DM32010 to 32019
LD Ok_Bit  ; Range Check OK Bit
OUT TR0
AND=(300) #BBBB UnitSelect  ; Specify the connetcted Unit SCB=#BBBB_SCU=&0to&15
MOVR(560) Type_D IR2  ; Address type DM start address
+L(401) IR2 &32000 IR2
LD TR0
AND<>(305) #BBBB UnitSelect  ; Specify the connetcted Unit SCB=#BBBB_SCU=&0to&15
AND<>(305) #CCCC UnitSelect  ; Specify the connetcted Unit SCB=#BBBB_SCU=&0to&15
MOVR(560) Type_D IR2  ; Address type DM start address
+L(401) IR2 &30000 IR2
*(420) UnitSelect &100 Offset  ; Specify the connetcted Unit SCB=#BBBB_SCU=&0to&15, For Address Culcurate
+L(401) IR2 Offset IR2  ; For Address Culcurate
LD TR0
AND<>(305) #CCCC UnitSelect  ; Specify the connetcted Unit SCB=#BBBB_SCU=&0to&15
AND=(300) &2 PortNo  ; Serial port No. &0to&2
+L(401) IR2 &10 IR2

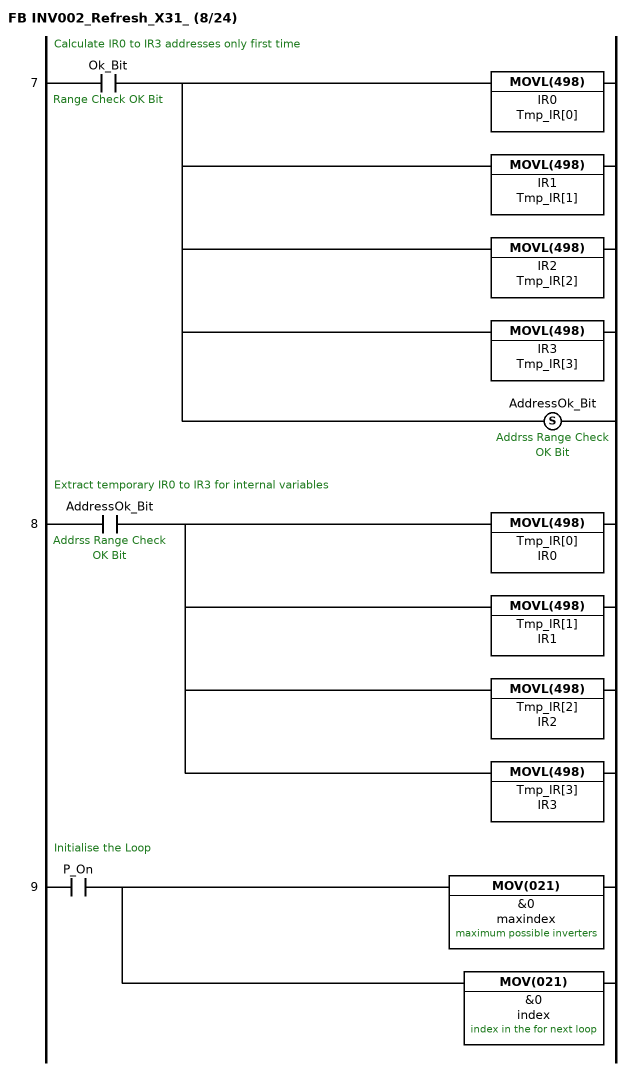
; rung 7: Calculate IR0 to IR3 addresses only first time
LD Ok_Bit  ; Range Check OK Bit
MOVL(498) IR0 Tmp_IR[0]
MOVL(498) IR1 Tmp_IR[1]
MOVL(498) IR2 Tmp_IR[2]
MOVL(498) IR3 Tmp_IR[3]
SET AddressOk_Bit  ; Addrss Range Check OK Bit
; rung 8: Extract temporary IR0 to IR3 for internal variables
LD AddressOk_Bit  ; Addrss Range Check OK Bit
MOVL(498) Tmp_IR[0] IR0
MOVL(498) Tmp_IR[1] IR1
MOVL(498) Tmp_IR[2] IR2
MOVL(498) Tmp_IR[3] IR3
; rung 9: Initialise the Loop
LD P_On
MOV(021) &0 maxindex  ; maximum possible inverters
MOV(021) &0 index  ; index in the for next loop

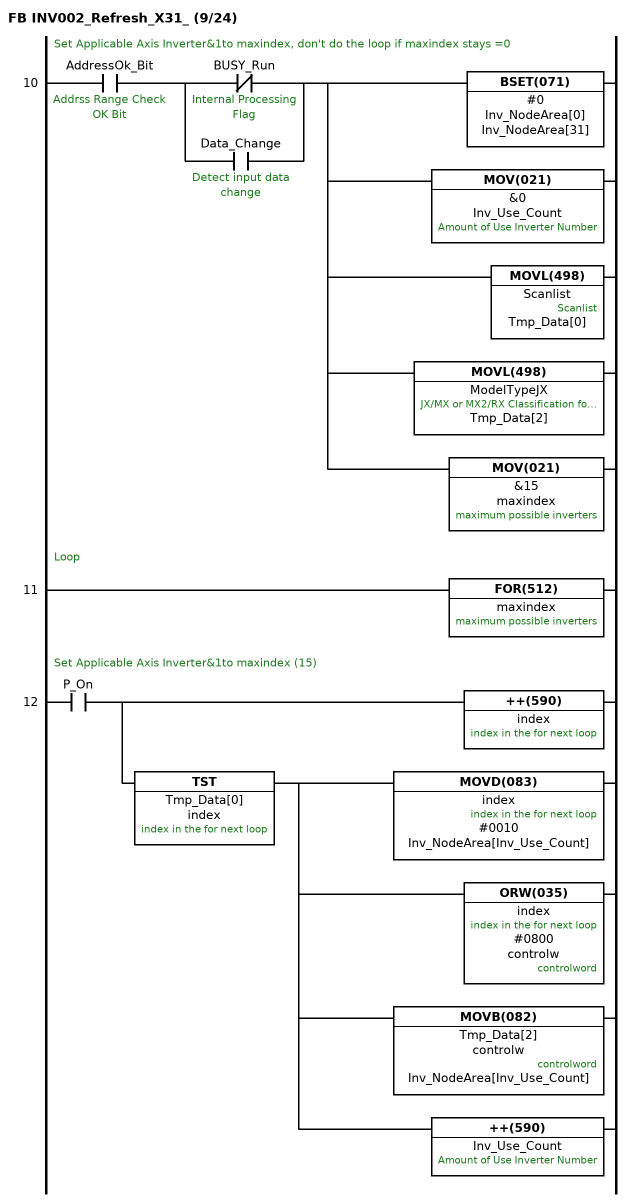
; rung 10: Set Applicable Axis Inverter&1to maxindex, don't do the loop if maxindex stays =0
LD AddressOk_Bit  ; Addrss Range Check OK Bit
LDNOT BUSY_Run  ; Internal Processing Flag
OR Data_Change  ; Detect input data change
ANDLD
BSET(071) #0 Inv_NodeArea[0] Inv_NodeArea[31]
MOV(021) &0 Inv_Use_Count  ; Amount of Use Inverter Number
MOVL(498) Scanlist Tmp_Data[0]  ; Scanlist
MOVL(498) ModelTypeJX Tmp_Data[2]  ; JX/MX or MX2/RX Classification for older Inverter types also this Bit has to be set, like scanlist
MOV(021) &15 maxindex  ; maximum possible inverters
; rung 11: Loop
FOR(512) maxindex  ; maximum possible inverters
; rung 12: Set Applicable Axis Inverter&1to maxindex (15)
LD P_On
++(590) index  ; index in the for next loop
ANDTST(350) Tmp_Data[0] index  ; index in the for next loop
MOVD(083) index #0010 Inv_NodeArea[Inv_Use_Count]  ; index in the for next loop
ORW(035) index #0800 controlw  ; index in the for next loop, controlword
MOVB(082) Tmp_Data[2] controlw Inv_NodeArea[Inv_Use_Count]  ; controlword
++(590) Inv_Use_Count  ; Amount of Use Inverter Number

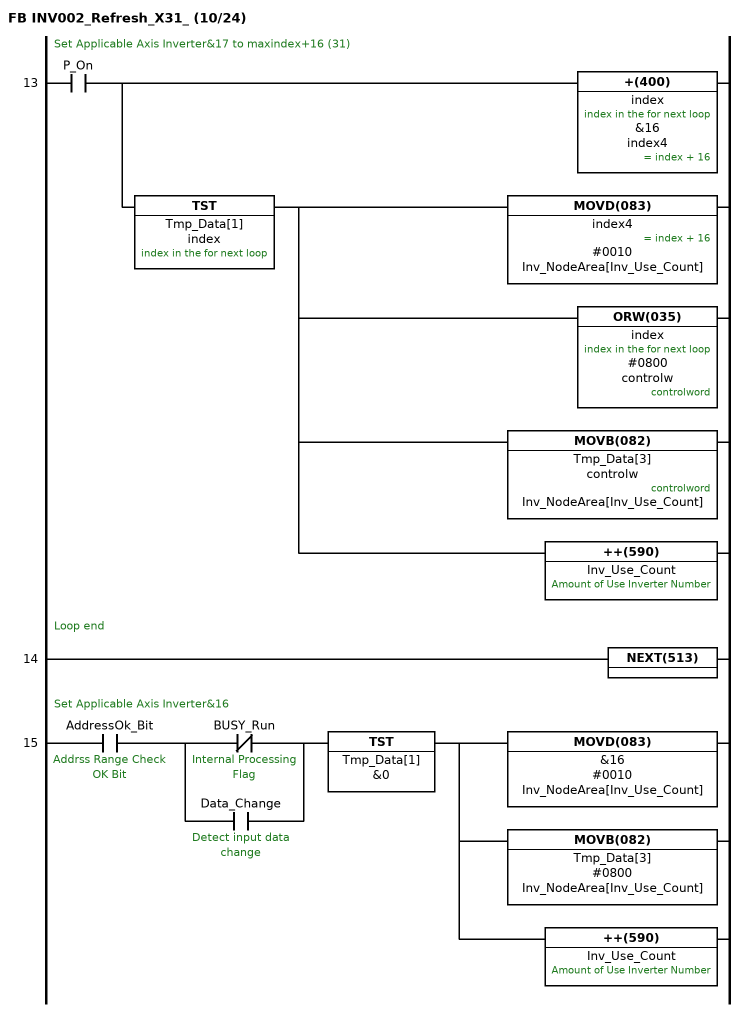
; rung 13: Set Applicable Axis Inverter&17 to maxindex+16 (31)
LD P_On
+(400) index &16 index4  ; index in the for next loop, = index + 16
ANDTST(350) Tmp_Data[1] index  ; index in the for next loop
MOVD(083) index4 #0010 Inv_NodeArea[Inv_Use_Count]  ; = index + 16
ORW(035) index #0800 controlw  ; index in the for next loop, controlword
MOVB(082) Tmp_Data[3] controlw Inv_NodeArea[Inv_Use_Count]  ; controlword
++(590) Inv_Use_Count  ; Amount of Use Inverter Number
; rung 14: Loop end
NEXT(513)
; rung 15: Set Applicable Axis Inverter&16
LD AddressOk_Bit  ; Addrss Range Check OK Bit
LDNOT BUSY_Run  ; Internal Processing Flag
OR Data_Change  ; Detect input data change
ANDLD
ANDTST(350) Tmp_Data[1] &0
MOVD(083) &16 #0010 Inv_NodeArea[Inv_Use_Count]
MOVB(082) Tmp_Data[3] #0800 Inv_NodeArea[Inv_Use_Count]
++(590) Inv_Use_Count  ; Amount of Use Inverter Number

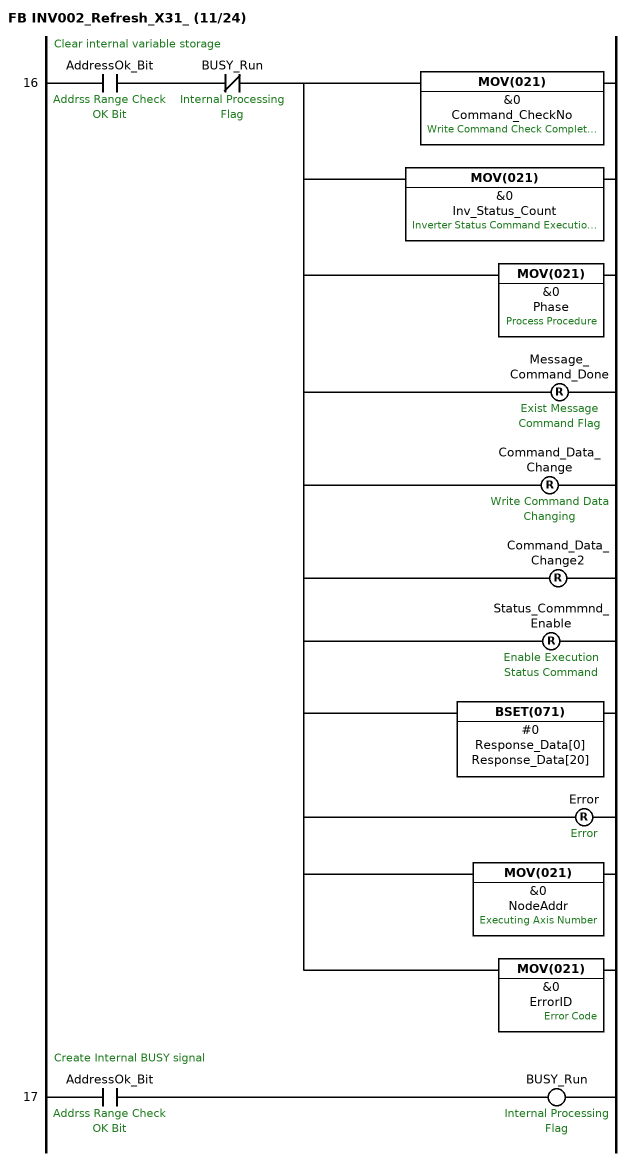
; rung 16: Clear internal variable storage
LD AddressOk_Bit  ; Addrss Range Check OK Bit
ANDNOT BUSY_Run  ; Internal Processing Flag
MOV(021) &0 Command_CheckNo  ; Write Command Check Complete Number
MOV(021) &0 Inv_Status_Count  ; Inverter Status Command Execution Number
MOV(021) &0 Phase  ; Process Procedure
RSET Message_Command_Done  ; Exist Message Command Flag
RSET Command_Data_Change  ; Write Command Data Changing
RSET Command_Data_Change2
RSET Status_Commmnd_Enable  ; Enable Execution Status Command
BSET(071) #0 Response_Data[0] Response_Data[20]
RSET Error  ; Error
MOV(021) &0 NodeAddr  ; Executing Axis Number
MOV(021) &0 ErrorID  ; Error Code
; rung 17: Create Internal BUSY signal
LD AddressOk_Bit  ; Addrss Range Check OK Bit
OUT BUSY_Run  ; Internal Processing Flag

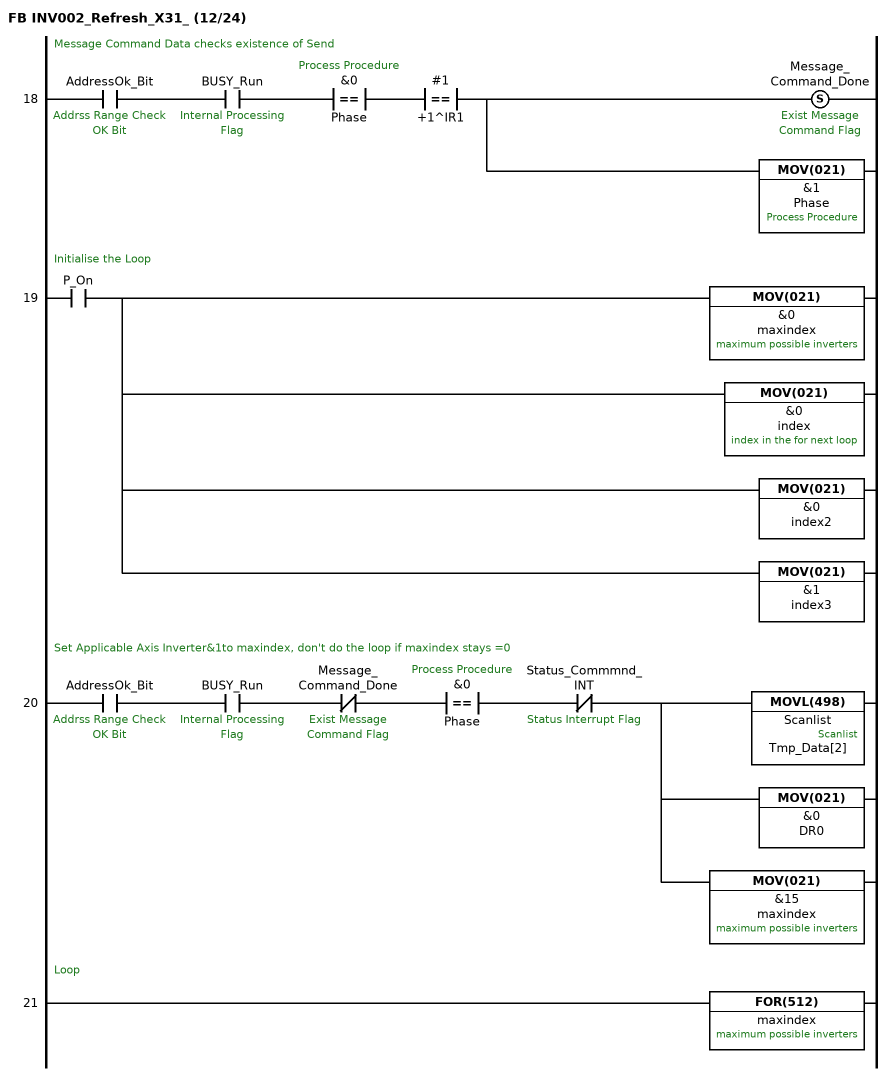
; rung 18: Message Command Data checks existence of Send
LD AddressOk_Bit  ; Addrss Range Check OK Bit
AND BUSY_Run  ; Internal Processing Flag
AND=(300) &0 Phase  ; Process Procedure
AND=(300) #1 +1^IR1
SET Message_Command_Done  ; Exist Message Command Flag
MOV(021) &1 Phase  ; Process Procedure
; rung 19: Initialise the Loop
LD P_On
MOV(021) &0 maxindex  ; maximum possible inverters
MOV(021) &0 index  ; index in the for next loop
MOV(021) &0 index2
MOV(021) &1 index3
; rung 20: Set Applicable Axis Inverter&1to maxindex, don't do the loop if maxindex stays =0
LD AddressOk_Bit  ; Addrss Range Check OK Bit
AND BUSY_Run  ; Internal Processing Flag
ANDNOT Message_Command_Done  ; Exist Message Command Flag
AND=(300) &0 Phase  ; Process Procedure
ANDNOT Status_Commmnd_INT  ; Status Interrupt Flag
MOVL(498) Scanlist Tmp_Data[2]  ; Scanlist
MOV(021) &0 DR0
MOV(021) &15 maxindex  ; maximum possible inverters
; rung 21: Loop
FOR(512) maxindex  ; maximum possible inverters

